Universal Robots URScript: RingModstack.script

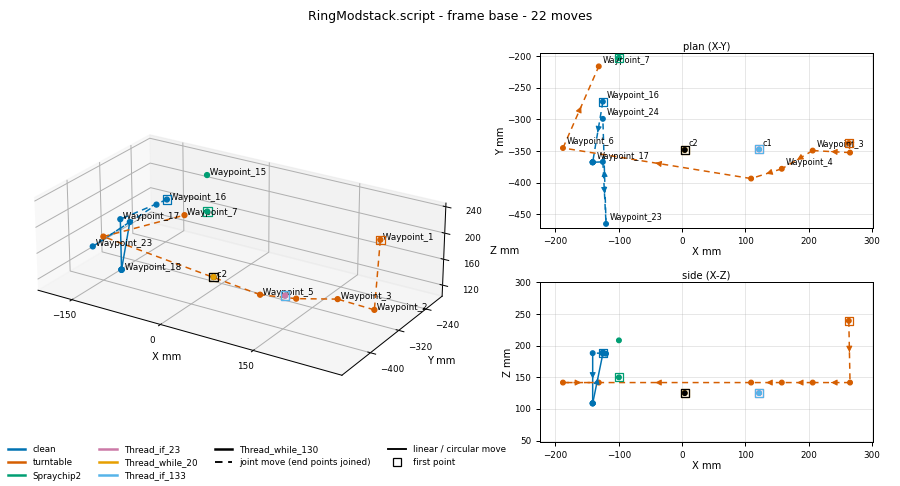
[picture p0: tool path of RingModstack.script in frame base, 22 of 62 moves have a stored position in this frame; points joined in program order, loops and branches not executed]
def RingModstack():
  global _hidden_verificationVariable=0
  step_count_fb48d3ff_0c9f_4d99_a765_ea41926c28d5 = 0.0
  thread Step_Counter_Thread_a9617a2c_6c0b_4ca4_aaba_c79477845290():
    while (True):
      step_count_fb48d3ff_0c9f_4d99_a765_ea41926c28d5 = step_count_fb48d3ff_0c9f_4d99_a765_ea41926c28d5 + 1.0
      sync()
    end
  end
  run Step_Counter_Thread_a9617a2c_6c0b_4ca4_aaba_c79477845290()
  set_standard_analog_input_domain(0, 1)
  set_standard_analog_input_domain(1, 1)
  set_tool_analog_input_domain(0, 1)
  set_tool_analog_input_domain(1, 1)
  set_analog_outputdomain(0, 0)
  set_analog_outputdomain(1, 0)
  set_input_actions_to_default()
  set_tool_communication(False, 115200, 0, 1, 1.5, 3.5)
  set_tool_output_mode(0)
  set_tool_digital_output_mode(0, 1)
  set_tool_digital_output_mode(1, 1)
  set_tool_voltage(0)
  set_safety_mode_transition_hardness(1)
  set_gravity([0.0, 0.0, 9.82])
  set_target_payload(0.530000, [0.009000, -0.039000, 0.092000], [0.000534, 0.000534, 0.000534, 0.000000, 0.000000, 0.000000])
  set_tcp(p[0.0,0.0,0.11,0.0,0.0,0.0])
  global Al_plate=p[0.12405209206180495,-0.2666666051843552,0.020008101224669964,-9.276623980477388E-5,1.8107917580596192E-5,3.1233857134705927]
  global Frame2x2=p[0.18266245434305164,-0.34273121659514855,0.026002571110600767,-2.225423529876215E-4,3.0110667546023537E-4,3.1233976058306383]
  global Plane_1=p[0.0,0.0,0.0,0.0,0.0,0.0]
  global URlogoTutorial=p[-0.08178353973148575,-0.3363174165299142,0.04788621506469384,-3.9746155723688456E-5,-3.4682148779121894E-5,-1.5668291789091222]
  global carousel=p[0.13865255139760183,-0.25132593351268107,0.051531504137083003,-4.453572132438073E-5,-1.3071222590669835E-4,-3.1349676625391965]
  global carouselrod=p[0.2020731702281844,-0.34951442511341274,0.1947611446273096,3.139766958234101,-0.10689428010274801,-1.1796370330365635E-5]
  global paper=p[-0.09670794781244417,-0.3283412964648025,0.027665994240809913,-3.2057893450593004E-5,2.867088716161181E-5,-1.6085327915291054]
  global rod=p[0.13368013097420872,-0.41123185103490206,0.09926814901395645,2.2214229924093103,-2.2214158162465862,-2.9165882738638143E-5]
  global timer_1=0
  global c1_p=p[.121821743145, -.347422555897, .125123580740, -3.141018983654, .028381750653, .002982050413]
  global c1_q=[-0.8683379332171839, -1.7976671657957972, -1.6403415203094482, -1.2751955848983307, 1.5710655450820923, 3.8608970642089844]
  global c2_p=p[.004287788739, -.348206668271, .125128550674, -3.141128603775, .028473860382, .002709910838]
  global c2_q=[-1.171152416859762, -1.712642332116598, -1.7442011833190918, -1.2557763022235413, 1.5706896781921387, 3.5581798553466797]
  global Waypoint_16_p=p[-.125097928533, -.271984222044, .188211676824, -3.139810722578, .105446315311, .000070958927]
  global Waypoint_16_q=[-1.5480602423297327, -1.4491210740855713, -1.7099264860153198, -1.552596167927124, 1.5715936422348022, 3.23006010055542]
  global Waypoint_17_p=p[-.141183217597, -.367684006591, .188213447751, 3.139821760490, -.105397104768, -.000067867997]
  global Waypoint_17_q=[-1.597567383443014, -1.8740092716612757, -1.241610050201416, -1.5960084400572718, 1.5719740390777588, 3.1803600788116455]
  global Waypoint_18_p=p[-.141178244459, -.367687282910, .108904454765, 3.139816402425, -.105408093734, -.000060814483]
  global Waypoint_18_q=[-1.5975983778582972, -1.9245020351805628, -1.550661325454712, -1.2364590925029297, 1.5723340511322021, 3.1807193756103516]
  global Waypoint_19_p=p[-.141189357305, -.367687267469, .108915260822, 3.121780755938, .351957921543, -.000099281586]
  global Waypoint_19_q=[-1.5976179281817835, -1.9244748554625453, -1.550661325454712, -1.2364507478526612, 1.572314977645874, 2.889045000076294]
  global Waypoint_20_p=p[-.141176698746, -.367682773595, .108907204798, -3.111042719163, .436975672702, .000063164110]
  global Waypoint_20_q=[-1.5975945631610315, -1.9244939289488734, -1.5506495237350464, -1.2365017098239441, 1.5723340511322021, 3.3926987648010254]
  global Waypoint_21_p=p[-.141174078526, -.367696805030, .108909057026, 3.139786221315, -.105395786134, -.000060564502]
  global Waypoint_21_q=[-1.597586456929342, -1.9245058498778285, -1.5506460666656494, -1.2364399594119568, 1.5723340511322021, 3.1807241439819336]
  global Waypoint_22_p=p[-.125093999497, -.367099400456, .187371407622, 3.139783011421, -.105392168035, -.000053869150]
  global Waypoint_22_q=[-1.5538747946368616, -1.846323629418844, -1.2822730541229248, -1.5829936466612757, 1.5719654560089111, 3.224064588546753]
  global Waypoint_23_p=p[-.120064390322, -.465070651334, .187365924664, 2.700279766902, -.088400420341, .019763045538]
  global Waypoint_23_q=[-1.5412524382220667, -1.9475652180113734, -1.406833291053772, -0.9173591893962403, 1.5603561401367188, 3.2332537174224854]
  global Waypoint_24_p=p[-.125099110421, -.299097154487, .189878767902, 3.139750209928, -.105401717856, -.000111797080]
  global Waypoint_24_q=[-1.550074879323141, -1.5617311683348198, -1.5979981422424316, -1.5518303674510499, 1.5716702938079834, 3.2279696464538574]
  global Waypoint_1_p=p[.263501689877, -.337317763427, .239349489480, 3.139797243720, -.105347053477, -.000037720516]
  global Waypoint_1_q=[-0.5959728399859827, -2.1057659588255824, -0.6533136367797852, -1.9525557957091273, 1.5718059539794922, 4.181682586669922]
  global Waypoint_2_p=p[.265438435610, -.352444474661, .141740907029, 3.139726376264, -.105360108121, -.000022031768]
  global Waypoint_2_q=[-0.6231134573565882, -2.1016999683775843, -1.126999020576477, -1.4828875821879883, 1.5722739696502686, 4.154912948608398]
  global Waypoint_3_p=p[.206441973084, -.349241721273, .141737893294, 3.139734184252, -.105329347268, -.000022485776]
  global Waypoint_3_q=[-0.7073677221881312, -1.9410401783385218, -1.3681066036224365, -1.4024366003325959, 1.5721865892410278, 4.070710182189941]
  global Waypoint_4_p=p[.157616611756, -.378012026932, .141738203587, 3.139764187573, -.105376653239, -.000076760662]
  global Waypoint_4_q=[-0.8494070211993616, -1.9579774341978968, -1.3439116477966309, -1.409730003481247, 1.5722019672393799, 3.928692579269409]
  global Waypoint_5_p=p[.109134761588, -.393436595889, .141742225598, 3.139732501163, -.105376381431, -.000050533951]
  global Waypoint_5_q=[-0.972816292439596, -1.9523960552611292, -1.3519116640090942, -1.4072665137103577, 1.5721949338912964, 3.805286407470703]
  global Waypoint_6_p=p[-.188131250090, -.345166366147, .141750553976, 3.139727051239, -.105353578209, -.000024875816]
  global Waypoint_6_q=[-1.7293437162982386, -1.8864180050291957, -1.4439769983291626, -1.381135032778122, 1.572224736213684, 3.0487747192382812]
  global Waypoint_7_p=p[-.131564048097, -.216205376465, .141741700579, 3.139714533984, -.105382776464, -.000044168049]
  global Waypoint_7_q=[-1.572542969380514, -1.2417927545360108, -2.0833356380462646, -1.3863917154124756, 1.571577787399292, 3.2058310508728027]
  global chipC_p=p[-.099707323994, -.202959245441, .150002109265, 3.139626928947, -.105484189856, -.000184527064]
  global chipC_q=[-1.4084599653827112, -1.0837949079326172, -2.1300156116485596, -1.4976508778384705, 1.571241855621338, 3.369978427886963]
  global Waypoint_15_p=p[-.099704296715, -.202951379992, .208432580258, 3.139670120847, -.105426183766, -.000160358536]
  global Waypoint_15_q=[-1.4082286993609827, -1.099871740942337, -1.8470300436019897, -1.764597078362936, 1.5709946155548096, 3.369927167892456]
  global timer_1_is_counting=False
  thread Timer_Thread():
    while (True):
      if (timer_1_is_counting):
        timer_1 = timer_1 + get_steptime()
      end
      sync()
    end
  end
  run Timer_Thread()
  def CircleAllangles():
    $ 324 "CircleAllangles" "noBreak"
    $ 325 "p0≔p[c[0]+r,c[1],c[2],c[3],c[4],c[5]-1.5*A]"
    global p0=p[c[0]+r,c[1],c[2],c[3],c[4],c[5]-1.5*A]
    $ 326 "p45≔p[c[0]+0.71*r,c[1]+0.71*r,c[2],c[3]-A/1.1,c[4],c[5]-A/1.1]"
    global p45=p[c[0]+0.71*r,c[1]+0.71*r,c[2],c[3]-A/1.1,c[4],c[5]-A/1.1]
    $ 327 "p90≔p[c[0],c[1]+r,c[2],c[3]-A,c[4],c[5]]"
    global p90=p[c[0],c[1]+r,c[2],c[3]-A,c[4],c[5]]
    $ 328 "p135≔p[c[0]-0.71*r,c[1]+0.71*r,c[2],c[3]-A/1.1,c[4],c[5]+A/1.1]"
    global p135=p[c[0]-0.71*r,c[1]+0.71*r,c[2],c[3]-A/1.1,c[4],c[5]+A/1.1]
    $ 329 "p180≔p[c[0]-r,c[1],c[2],c[3],c[4],c[5]+1.5*A]"
    global p180=p[c[0]-r,c[1],c[2],c[3],c[4],c[5]+1.5*A]
    $ 330 "p225≔p[c[0]-0.71*r,c[1]-0.71*r,c[2],c[3]+A/1.1,c[4],c[5]+A/1.1]"
    global p225=p[c[0]-0.71*r,c[1]-0.71*r,c[2],c[3]+A/1.1,c[4],c[5]+A/1.1]
    $ 331 "p270≔p[c[0],c[1]-r,c[2],c[3]+A,c[4],c[5]]"
    global p270=p[c[0],c[1]-r,c[2],c[3]+A,c[4],c[5]]
    $ 332 "p315≔p[c[0]+0.71*r,c[1]-0.71*r,c[2],c[3]+A/1.1,c[4],c[5]-A/1.1]"
    global p315=p[c[0]+0.71*r,c[1]-0.71*r,c[2],c[3]+A/1.1,c[4],c[5]-A/1.1]
    $ 333 "Set atomization=On"
    set_standard_digital_out(1, True)
    $ 334 "Set triggersolenoid=On"
    set_standard_digital_out(0, True)
    $ 335 "MoveL"
    $ 336 "p0" "breakAfter"
    set_tcp(p[0.0,0.0,0.11,0.0,0.0,0.0])
    movel(p0, a=1.3, v=0.4, r=0.005)
    $ 337 "p45" "breakAfter"
    set_tcp(p[0.0,0.0,0.11,0.0,0.0,0.0])
    movel(p45, a=1.3, v=0.4, r=0.005)
    $ 338 "p90" "breakAfter"
    set_tcp(p[0.0,0.0,0.11,0.0,0.0,0.0])
    movel(p90, a=1.3, v=0.4, r=0.005)
    $ 339 "p135" "breakAfter"
    set_tcp(p[0.0,0.0,0.11,0.0,0.0,0.0])
    movel(p135, a=1.3, v=0.4, r=0.005)
    $ 340 "p180" "breakAfter"
    set_tcp(p[0.0,0.0,0.11,0.0,0.0,0.0])
    movel(p180, a=1.3, v=0.4, r=0.005)
    $ 341 "p225" "breakAfter"
    set_tcp(p[0.0,0.0,0.11,0.0,0.0,0.0])
    movel(p225, a=1.3, v=0.4, r=0.005)
    $ 342 "p270" "breakAfter"
    set_tcp(p[0.0,0.0,0.11,0.0,0.0,0.0])
    movel(p270, a=1.3, v=0.4, r=0.005)
    $ 343 "p315" "breakAfter"
    set_tcp(p[0.0,0.0,0.11,0.0,0.0,0.0])
    movel(p315, a=1.3, v=0.4, r=0.005)
    $ 344 "p0" "breakAfter"
    set_tcp(p[0.0,0.0,0.11,0.0,0.0,0.0])
    movel(p0, a=1.3, v=0.4, r=0.005)
    $ 345 "p45" "breakAfter"
    set_tcp(p[0.0,0.0,0.11,0.0,0.0,0.0])
    movel(p45, a=1.3, v=0.4, r=0.005)
    $ 346 "p90" "breakAfter"
    set_tcp(p[0.0,0.0,0.11,0.0,0.0,0.0])
    movel(p90, a=1.3, v=0.4, r=0.005)
    $ 347 "Set triggersolenoid=Off"
    set_standard_digital_out(0, False)
    $ 348 "Wait: 0.3"
    sleep(0.3)
    $ 349 "Set atomization=Off"
    set_standard_digital_out(1, False)
  end
  def clean():
    $ 350 "clean" "noBreak"
    $ 351 "MoveJ"
    $ 352 "Waypoint_16" "breakAfter"
    movej(get_inverse_kin(Waypoint_16_p, qnear=Waypoint_16_q), a=1.3962634015954636, v=1.0471975511965976)
    $ 353 "Waypoint_17" "breakAfter"
    movej(get_inverse_kin(Waypoint_17_p, qnear=Waypoint_17_q), a=1.3962634015954636, v=1.0471975511965976)
    $ 354 "MoveL"
    $ 355 "Waypoint_18" "breakAfter"
    movel(Waypoint_18_p, a=1.2, v=0.05)
    $ 356 "MoveL"
    $ 357 "Waypoint_19" "breakAfter"
    movel(Waypoint_19_p, a=1.2, v=0.05)
    $ 358 "MoveL"
    $ 359 "Waypoint_20" "breakAfter"
    movel(Waypoint_20_p, a=1.2, v=0.05)
    $ 360 "MoveL"
    $ 361 "Waypoint_21" "breakAfter"
    movel(Waypoint_21_p, a=1.2, v=0.05)
    $ 362 "MoveL"
    $ 363 "Waypoint_22" "breakAfter"
    movel(Waypoint_22_p, a=1.2, v=0.25)
    $ 364 "MoveJ"
    $ 365 "Waypoint_23" "breakAfter"
    movej(get_inverse_kin(Waypoint_23_p, qnear=Waypoint_23_q), a=1.3962634015954636, v=1.0471975511965976)
    $ 366 "Set atomization=On"
    set_standard_digital_out(1, True)
    $ 367 "Set triggersolenoid=On"
    set_standard_digital_out(0, True)
    $ 368 "Wait: 0.2"
    sleep(0.2)
    $ 369 "Set triggersolenoid=Off"
    set_standard_digital_out(0, False)
    $ 370 "Set atomization=Off"
    set_standard_digital_out(1, False)
    $ 371 "MoveJ"
    $ 372 "Waypoint_24" "breakAfter"
    movej(get_inverse_kin(Waypoint_24_p, qnear=Waypoint_24_q), a=1.3962634015954636, v=1.0471975511965976)
  end
  def turntable():
    $ 373 "turntable" "noBreak"
    $ 374 "MoveJ"
    $ 375 "Waypoint_1" "breakAfter"
    set_tcp(p[0.0,0.0,0.11,0.0,0.0,0.0])
    movej(get_inverse_kin(pose_trans(carouselrod, pose_trans(p[-.225374943892, -.334963115589, .194760490875, -3.139766958133, .106894280099, .000011796372], Waypoint_1_p)), qnear=Waypoint_1_q), a=1.3962634015954636, v=0.5235987755982988, r=0.02)
    $ 376 "Waypoint_2" "breakAfter"
    set_tcp(p[0.0,0.0,0.11,0.0,0.0,0.0])
    movej(get_inverse_kin(pose_trans(carouselrod, pose_trans(p[-.225374943892, -.334963115589, .194760490875, -3.139766958133, .106894280099, .000011796372], Waypoint_2_p)), qnear=Waypoint_2_q), a=1.3962634015954636, v=0.5235987755982988, r=0.02)
    $ 377 "Waypoint_3" "breakAfter"
    set_tcp(p[0.0,0.0,0.11,0.0,0.0,0.0])
    movej(get_inverse_kin(pose_trans(carouselrod, pose_trans(p[-.225374943892, -.334963115589, .194760490875, -3.139766958133, .106894280099, .000011796372], Waypoint_3_p)), qnear=Waypoint_3_q), a=1.3962634015954636, v=0.5235987755982988, r=0.02)
    $ 378 "Waypoint_4" "breakAfter"
    set_tcp(p[0.0,0.0,0.11,0.0,0.0,0.0])
    movej(get_inverse_kin(pose_trans(carouselrod, pose_trans(p[-.225374943892, -.334963115589, .194760490875, -3.139766958133, .106894280099, .000011796372], Waypoint_4_p)), qnear=Waypoint_4_q), a=1.3962634015954636, v=0.5235987755982988, r=0.02)
    $ 379 "Waypoint_5" "breakAfter"
    set_tcp(p[0.0,0.0,0.11,0.0,0.0,0.0])
    movej(get_inverse_kin(pose_trans(carouselrod, pose_trans(p[-.225374943892, -.334963115589, .194760490875, -3.139766958133, .106894280099, .000011796372], Waypoint_5_p)), qnear=Waypoint_5_q), a=1.3962634015954636, v=0.5235987755982988, r=0.02)
    $ 380 "MoveJ"
    $ 381 "Waypoint_6" "breakAfter"
    movej(get_inverse_kin(pose_trans(carouselrod, pose_trans(p[-.225374943892, -.334963115589, .194760490875, -3.139766958133, .106894280099, .000011796372], Waypoint_6_p)), qnear=Waypoint_6_q), a=1.3962634015954636, v=0.3141592653589793)
    $ 382 "Wait: 1.0"
    sleep(1.0)
    $ 383 "MoveJ"
    $ 384 "Waypoint_7" "breakAfter"
    movej(get_inverse_kin(pose_trans(carouselrod, pose_trans(p[-.225374943892, -.334963115589, .194760490875, -3.139766958133, .106894280099, .000011796372], Waypoint_7_p)), qnear=Waypoint_7_q), a=1.3962634015954636, v=1.0471975511965976, r=0.02)
  end
  def Spraychip2():
    $ 385 "Spraychip2" "noBreak"
    $ 386 "MoveJ"
    $ 387 "chipC" "breakAfter"
    movej(get_inverse_kin(chipC_p, qnear=chipC_q), a=1.3962634015954636, v=1.0471975511965976)
    $ 388 "c≔chipC"
    global c=chipC_p
    $ 389 "rc≔27/1000"
    global rc=27/1000
    $ 390 "p0≔p[c[0]+rc,c[1],c[2],c[3],c[4],c[5]-1.5*0]"
    global p0=p[c[0]+rc,c[1],c[2],c[3],c[4],c[5]-1.5*0]
    $ 391 "p45≔p[c[0]+0.71*rc,c[1]+0.71*rc,c[2],c[3]-0/1.1,c[4],c[5]-0/1.1]"
    global p45=p[c[0]+0.71*rc,c[1]+0.71*rc,c[2],c[3]-0/1.1,c[4],c[5]-0/1.1]
    $ 392 "p90≔p[c[0],c[1]+rc,c[2],c[3]-0,c[4],c[5]]"
    global p90=p[c[0],c[1]+rc,c[2],c[3]-0,c[4],c[5]]
    $ 393 "p135≔p[c[0]-0.71*rc,c[1]+0.71*rc,c[2],c[3]-0/1.1,c[4],c[5]+0/1.1]"
    global p135=p[c[0]-0.71*rc,c[1]+0.71*rc,c[2],c[3]-0/1.1,c[4],c[5]+0/1.1]
    $ 394 "p180≔p[c[0]-rc,c[1],c[2],c[3],c[4],c[5]+1.5*0]"
    global p180=p[c[0]-rc,c[1],c[2],c[3],c[4],c[5]+1.5*0]
    $ 395 "p225≔p[c[0]-0.71*rc,c[1]-0.71*rc,c[2],c[3]+0/1.1,c[4],c[5]+0/1.1]"
    global p225=p[c[0]-0.71*rc,c[1]-0.71*rc,c[2],c[3]+0/1.1,c[4],c[5]+0/1.1]
    $ 396 "p270≔p[c[0],c[1]-rc,c[2],c[3]+0,c[4],c[5]]"
    global p270=p[c[0],c[1]-rc,c[2],c[3]+0,c[4],c[5]]
    $ 397 "p315≔p[c[0]+0.71*rc,c[1]-0.71*rc,c[2],c[3]+0/1.1,c[4],c[5]-0/1.1]"
    global p315=p[c[0]+0.71*rc,c[1]-0.71*rc,c[2],c[3]+0/1.1,c[4],c[5]-0/1.1]
    $ 398 "Set atomization=On"
    set_standard_digital_out(1, True)
    $ 399 "Set triggersolenoid=On"
    set_standard_digital_out(0, True)
    $ 400 "MoveL"
    $ 401 "p0" "breakAfter"
    set_tcp(p[0.0,0.0,0.11,0.0,0.0,0.0])
    movel(p0, a=1.3, v=0.085, r=0.01)
    $ 402 "p45" "breakAfter"
    set_tcp(p[0.0,0.0,0.11,0.0,0.0,0.0])
    movel(p45, a=1.3, v=0.085, r=0.01)
    $ 403 "p90" "breakAfter"
    set_tcp(p[0.0,0.0,0.11,0.0,0.0,0.0])
    movel(p90, a=1.3, v=0.085, r=0.01)
    $ 404 "p135" "breakAfter"
    set_tcp(p[0.0,0.0,0.11,0.0,0.0,0.0])
    movel(p135, a=1.3, v=0.085, r=0.01)
    $ 405 "p180" "breakAfter"
    set_tcp(p[0.0,0.0,0.11,0.0,0.0,0.0])
    movel(p180, a=1.3, v=0.085, r=0.01)
    $ 406 "Set triggersolenoid=Off"
    set_standard_digital_out(0, False)
    $ 407 "Wait: 0.1"
    sleep(0.1)
    $ 408 "Set triggersolenoid=On"
    set_standard_digital_out(0, True)
    $ 409 "p225" "breakAfter"
    set_tcp(p[0.0,0.0,0.11,0.0,0.0,0.0])
    movel(p225, a=1.3, v=0.085, r=0.01)
    $ 410 "p270" "breakAfter"
    set_tcp(p[0.0,0.0,0.11,0.0,0.0,0.0])
    movel(p270, a=1.3, v=0.085, r=0.01)
    $ 411 "p315" "breakAfter"
    set_tcp(p[0.0,0.0,0.11,0.0,0.0,0.0])
    movel(p315, a=1.3, v=0.085, r=0.01)
    $ 412 "p0" "breakAfter"
    set_tcp(p[0.0,0.0,0.11,0.0,0.0,0.0])
    movel(p0, a=1.3, v=0.085, r=0.01)
    $ 413 "p45" "breakAfter"
    set_tcp(p[0.0,0.0,0.11,0.0,0.0,0.0])
    movel(p45, a=1.3, v=0.085, r=0.01)
    $ 414 "Set triggersolenoid=Off"
    set_standard_digital_out(0, False)
    $ 415 "Wait: 0.1"
    sleep(0.1)
    $ 416 "Set triggersolenoid=On"
    set_standard_digital_out(0, True)
    $ 417 "p90" "breakAfter"
    set_tcp(p[0.0,0.0,0.11,0.0,0.0,0.0])
    movel(p90, a=1.3, v=0.085, r=0.01)
    $ 418 "p135" "breakAfter"
    set_tcp(p[0.0,0.0,0.11,0.0,0.0,0.0])
    movel(p135, a=1.3, v=0.085, r=0.01)
    $ 419 "p180" "breakAfter"
    set_tcp(p[0.0,0.0,0.11,0.0,0.0,0.0])
    movel(p180, a=1.3, v=0.085, r=0.01)
    $ 420 "p225" "breakAfter"
    set_tcp(p[0.0,0.0,0.11,0.0,0.0,0.0])
    movel(p225, a=1.3, v=0.085, r=0.01)
    $ 421 "p270" "breakAfter"
    set_tcp(p[0.0,0.0,0.11,0.0,0.0,0.0])
    movel(p270, a=1.3, v=0.085, r=0.01)
    $ 422 "p315" "breakAfter"
    set_tcp(p[0.0,0.0,0.11,0.0,0.0,0.0])
    movel(p315, a=1.3, v=0.085, r=0.01)
    $ 423 "p0" "breakAfter"
    set_tcp(p[0.0,0.0,0.11,0.0,0.0,0.0])
    movel(p0, a=1.3, v=0.085, r=0.01)
    $ 424 "MoveJ"
    $ 425 "Waypoint_15" "breakAfter"
    movej(get_inverse_kin(Waypoint_15_p, qnear=Waypoint_15_q), a=1.3962634015954636, v=1.0471975511965976)
    $ 426 "Wait: 0.2"
    sleep(0.2)
    $ 427 "Set triggersolenoid=Off"
    set_standard_digital_out(0, False)
    $ 428 "Wait: 0.3"
    sleep(0.3)
    $ 429 "Set atomization=Off"
    set_standard_digital_out(1, False)
  end
  while (True):
    $ 2 "Robot Program"
    $ 3 "'Program to be used for part #124517-043 lens ring mod when stacked'"
    # 'Program to be used for part #124517-043 lens ring mod when stacked'
    $ 4 "'Program rev A: 8/26/24 adjusted spray centers to corrected positions for new(?) masks'"
    # 'Program rev A: 8/26/24 adjusted spray centers to corrected positions for new(?) masks'
    $ 5 "timer_1: Start"
    timer_1_is_counting = True
    $ 6 "r≔1/1000"
    global r=1/1000
    $ 7 "A≔8*3.1416/180"
    global A=8*3.1416/180
    $ 10 "Loop_1≔1"
    global Loop_1=1
    $ 11 "sidenum≔2"
    global sidenum=2
    $ 13 "partnum≔3"
    global partnum=3
    $ 15 "coatnum≔2"
    global coatnum=2
    $ 16 "If partnum≤sidenum"
    global thread_flag_16=0
    thread Thread_if_16():
      $ 17 "Loop (coatnum)>0"
      thread Thread_while_17():
        while (True):
          $ 18 "partleft≔partnum"
          global partleft=partnum
          $ 19 "loopnum≔1"
          global loopnum=1
          $ 20 "Loop partleft>0"
          thread Thread_while_20():
            while (True):
              $ 21 "Call clean"
              clean()
              $ 22 "Call Spraychip2"
              Spraychip2()
              $ 23 "If loopnum≟1 or loopnum≟3 or loopnum≟5 or loopnum≟7 or loopnum≟9 or loopnum≟11"
              global thread_flag_23=0
              thread Thread_if_23():
                $ 53 "MoveJ"
                $ 54 "c1" "breakAfter"
                movej(get_inverse_kin(c1_p, qnear=c1_q), a=1.3962634015954636, v=1.0471975511965976)
                $ 55 "c≔c1"
                global c=c1_p
                $ 56 "Call CircleAllangles"
                CircleAllangles()
                $ 57 "x2≔p[c[0]-0.051,c[1],c[2],c[3],c[4],c[5]]"
                global x2=p[c[0]-0.051,c[1],c[2],c[3],c[4],c[5]]
                $ 58 "x3≔p[c[0]-0.051,c[1]+0.051,c[2],c[3],c[4],c[5]]"
                global x3=p[c[0]-0.051,c[1]+0.051,c[2],c[3],c[4],c[5]]
                $ 59 "x4≔p[c[0],c[1]+0.051,c[2],c[3],c[4],c[5]]"
                global x4=p[c[0],c[1]+0.051,c[2],c[3],c[4],c[5]]
                $ 60 "MoveJ"
                $ 61 "x2" "breakAfter"
                movej(x2, a=1.3962634015954636, v=1.0471975511965976)
                $ 62 "c≔x2"
                global c=x2
                $ 63 "Call CircleAllangles"
                CircleAllangles()
                $ 64 "MoveJ"
                $ 65 "x3" "breakAfter"
                movej(x3, a=1.3962634015954636, v=1.0471975511965976)
                $ 66 "c≔x3"
                global c=x3
                $ 67 "Call CircleAllangles"
                CircleAllangles()
                $ 68 "MoveJ"
                $ 69 "x4" "breakAfter"
                movej(x4, a=1.3962634015954636, v=1.0471975511965976)
                $ 70 "c≔x4"
                global c=x4
                $ 71 "Call CircleAllangles"
                CircleAllangles()
                thread_flag_23 = 1
              end
              if (loopnum == 1  or  loopnum == 3  or  loopnum == 5  or  loopnum == 7  or  loopnum == 9  or  loopnum == 11):
                global thread_handler_23=run Thread_if_23()
                while (thread_flag_23 == 0):
                  if not(loopnum == 1  or  loopnum == 3  or  loopnum == 5  or  loopnum == 7  or  loopnum == 9  or  loopnum == 11):
                    kill thread_handler_23
                    thread_flag_23 = 2
                  else:
                    sync()
                  end
                end
              else:
                thread_flag_23 = 2
              end
              if (thread_flag_23 == 2):
                $ 72 "Else" "noBreak"
                $ 101 "MoveJ"
                $ 102 "c2" "breakAfter"
                movej(get_inverse_kin(c2_p, qnear=c2_q), a=1.3962634015954636, v=1.0471975511965976)
                $ 103 "c≔c2"
                global c=c2_p
                $ 104 "Call CircleAllangles"
                CircleAllangles()
                $ 105 "x2≔p[c[0]-0.051,c[1],c[2],c[3],c[4],c[5]]"
                global x2=p[c[0]-0.051,c[1],c[2],c[3],c[4],c[5]]
                $ 106 "x3≔p[c[0]-0.051,c[1]+0.051,c[2],c[3],c[4],c[5]]"
                global x3=p[c[0]-0.051,c[1]+0.051,c[2],c[3],c[4],c[5]]
                $ 107 "x4≔p[c[0],c[1]+0.051,c[2],c[3],c[4],c[5]]"
                global x4=p[c[0],c[1]+0.051,c[2],c[3],c[4],c[5]]
                $ 108 "MoveJ"
                $ 109 "x2" "breakAfter"
                movej(x2, a=1.3962634015954636, v=1.0471975511965976)
                $ 110 "c≔x2"
                global c=x2
                $ 111 "Call CircleAllangles"
                CircleAllangles()
                $ 112 "MoveJ"
                $ 113 "x3" "breakAfter"
                movej(x3, a=1.3962634015954636, v=1.0471975511965976)
                $ 114 "c≔x3"
                global c=x3
                $ 115 "Call CircleAllangles"
                CircleAllangles()
                $ 116 "MoveJ"
                $ 117 "x4" "breakAfter"
                movej(x4, a=1.3962634015954636, v=1.0471975511965976)
                $ 118 "c≔x4"
                global c=x4
                $ 119 "Call CircleAllangles"
                CircleAllangles()
              end
              $ 120 "loopnum≔loopnum+1"
              global loopnum=loopnum+1
              $ 121 "partleft≔partleft-1"
              global partleft=partleft-1
            end
          end
          if (partleft>0):
            global thread_handler_20=run Thread_while_20()
            while (partleft>0):
              sync()
            end
            kill thread_handler_20
          end
          $ 122 "i≔0"
          global i=0
          $ 123 "coatnum≔coatnum-1"
          global coatnum=coatnum-1
        end
      end
      if ((coatnum)>0):
        global thread_handler_17=run Thread_while_17()
        while ((coatnum)>0):
          sync()
        end
        kill thread_handler_17
      end
      $ 124 "Halt"
      halt
      thread_flag_16 = 1
    end
    if (partnum <= sidenum):
      global thread_handler_16=run Thread_if_16()
      while (thread_flag_16 == 0):
        if not(partnum <= sidenum):
          kill thread_handler_16
          thread_flag_16 = 2
        else:
          sync()
        end
      end
    else:
      thread_flag_16 = 2
    end
    if (thread_flag_16 == 2):
      $ 125 "Else" "noBreak"
      $ 126 "Loop (coatnum)>0"
      thread Thread_while_126():
        while (True):
          $ 127 "partleft≔partnum"
          global partleft=partnum
          $ 128 "loopnum≔1"
          global loopnum=1
          $ 129 "turnnum≔0"
          global turnnum=0
          $ 130 "Loop partleft>0"
          thread Thread_while_130():
            while (True):
              $ 131 "Call clean"
              clean()
              $ 132 "Call Spraychip2"
              Spraychip2()
              $ 133 "If loopnum≟1 or loopnum≟3 or loopnum≟5 or loopnum≟7 or loopnum≟9 or loopnum≟11"
              global thread_flag_133=0
              thread Thread_if_133():
                $ 163 "MoveJ"
                $ 164 "c1" "breakAfter"
                movej(get_inverse_kin(c1_p, qnear=c1_q), a=1.3962634015954636, v=1.0471975511965976)
                $ 165 "c≔c1"
                global c=c1_p
                $ 166 "Call CircleAllangles"
                CircleAllangles()
                $ 167 "x2≔p[c[0]-0.051,c[1],c[2],c[3],c[4],c[5]]"
                global x2=p[c[0]-0.051,c[1],c[2],c[3],c[4],c[5]]
                $ 168 "x3≔p[c[0]-0.051,c[1]+0.051,c[2],c[3],c[4],c[5]]"
                global x3=p[c[0]-0.051,c[1]+0.051,c[2],c[3],c[4],c[5]]
                $ 169 "x4≔p[c[0],c[1]+0.051,c[2],c[3],c[4],c[5]]"
                global x4=p[c[0],c[1]+0.051,c[2],c[3],c[4],c[5]]
                $ 170 "MoveJ"
                $ 171 "x2" "breakAfter"
                movej(x2, a=1.3962634015954636, v=1.0471975511965976)
                $ 172 "c≔x2"
                global c=x2
                $ 173 "Call CircleAllangles"
                CircleAllangles()
                $ 174 "MoveJ"
                $ 175 "x3" "breakAfter"
                movej(x3, a=1.3962634015954636, v=1.0471975511965976)
                $ 176 "c≔x3"
                global c=x3
                $ 177 "Call CircleAllangles"
                CircleAllangles()
                $ 178 "MoveJ"
                $ 179 "x4" "breakAfter"
                movej(x4, a=1.3962634015954636, v=1.0471975511965976)
                $ 180 "c≔x4"
                global c=x4
                $ 181 "Call CircleAllangles"
                CircleAllangles()
                thread_flag_133 = 1
              end
              if (loopnum == 1  or  loopnum == 3  or  loopnum == 5  or  loopnum == 7  or  loopnum == 9  or  loopnum == 11):
                global thread_handler_133=run Thread_if_133()
                while (thread_flag_133 == 0):
                  if not(loopnum == 1  or  loopnum == 3  or  loopnum == 5  or  loopnum == 7  or  loopnum == 9  or  loopnum == 11):
                    kill thread_handler_133
                    thread_flag_133 = 2
                  else:
                    sync()
                  end
                end
              else:
                thread_flag_133 = 2
              end
              if (thread_flag_133 == 2):
                $ 182 "Else" "noBreak"
                $ 213 "MoveJ"
                $ 214 "c2" "breakAfter"
                movej(get_inverse_kin(c2_p, qnear=c2_q), a=1.3962634015954636, v=1.0471975511965976)
                $ 215 "c≔c2"
                global c=c2_p
                $ 216 "Call CircleAllangles"
                CircleAllangles()
                $ 217 "x2≔p[c[0]-0.051,c[1],c[2],c[3],c[4],c[5]]"
                global x2=p[c[0]-0.051,c[1],c[2],c[3],c[4],c[5]]
                $ 218 "x3≔p[c[0]-0.051,c[1]+0.051,c[2],c[3],c[4],c[5]]"
                global x3=p[c[0]-0.051,c[1]+0.051,c[2],c[3],c[4],c[5]]
                $ 219 "x4≔p[c[0],c[1]+0.051,c[2],c[3],c[4],c[5]]"
                global x4=p[c[0],c[1]+0.051,c[2],c[3],c[4],c[5]]
                $ 220 "MoveJ"
                $ 221 "x2" "breakAfter"
                movej(x2, a=1.3962634015954636, v=1.0471975511965976)
                $ 222 "c≔x2"
                global c=x2
                $ 223 "Call CircleAllangles"
                CircleAllangles()
                $ 224 "MoveJ"
                $ 225 "x3" "breakAfter"
                movej(x3, a=1.3962634015954636, v=1.0471975511965976)
                $ 226 "c≔x3"
                global c=x3
                $ 227 "Call CircleAllangles"
                CircleAllangles()
                $ 228 "MoveJ"
                $ 229 "x4" "breakAfter"
                movej(x4, a=1.3962634015954636, v=1.0471975511965976)
                $ 230 "c≔x4"
                global c=x4
                $ 231 "Call CircleAllangles"
                CircleAllangles()
              end
              $ 232 "loopnum≔loopnum+1"
              global loopnum=loopnum+1
              $ 233 "partleft≔partleft-1"
              global partleft=partleft-1
            end
          end
          if (partleft>0):
            global thread_handler_130=run Thread_while_130()
            while (partleft>0):
              sync()
            end
            kill thread_handler_130
          end
          $ 234 "i≔0"
          global i=0
          $ 235 "Loop (6-turnnum)>0"
          thread Thread_while_235():
            while (True):
              $ 236 "Call turntable"
              turntable()
              $ 237 "turnnum≔turnnum+1"
              global turnnum=turnnum+1
            end
          end
          if ((6-turnnum)>0):
            global thread_handler_235=run Thread_while_235()
            while ((6-turnnum)>0):
              sync()
            end
            kill thread_handler_235
          end
          $ 238 "coatnum≔coatnum-1"
          global coatnum=coatnum-1
        end
      end
      if ((coatnum)>0):
        global thread_handler_126=run Thread_while_126()
        while ((coatnum)>0):
          sync()
        end
        kill thread_handler_126
      end
      $ 239 "Halt"
      halt
    end
  end
end
